Staubli VAL3: getPwrCnt.pgx

program getPwrCnt()
begin
  //
  nPwrCnt=$getPowerCount()
  gotoxy(1,8)
  put("总上电小时数："+toString("",nPwrCnt))
end
